// TIA Portal V20 export
FUNCTION_BLOCK "AirConditioner"   // FB349, FBD
{ S7_Optimized_Access := 'TRUE' }
// stored: AutoNumber false, MemoryReserve 100, SetENOAutomatically false
   VAR
      Var : "TypeVar";
      T : Array[1..4] of IEC_TIMER;
   END_VAR
   VAR DB_SPECIFIC
      air1Active : Bool := 1;   // air conditioner 1 scannerhousing visual measurement active
      air1InputNo : Bool := 0;   // air conditioner 1 scannerhousing visual measurement input normal
      air2Active : Bool := 1;   // air conditioner 2 scannerhousing visual measurement active
      air2InputNo : Bool := 0;   // air conditioner 2 scannerhousing visual measurement input normal
      airXrayActive : Bool := 1;   // air conditioner scannerhousing x-ray measurement active
      airXrayInputNo : Bool := 0;   // air conditioner scannerhousing x-ray measurement input normal
      airDehActive : Bool := 0;   // air dehumidifier active
      airDehInputNo : Bool := 0;   // air dehumidifier input normal open
   END_VAR
BEGIN

REGION Network 1 (SCL): air conditioner 1&2 visual measurement - config from Pc
   "G".air1Off := INT_TO_BOOL( "Param".Rd.air1Off);
   "G".air2Off := INT_TO_BOOL("Param".Rd.air2Off);
   #air1Active := INT_TO_BOOL("Param".Rd.air1Active);
   #air2Active := INT_TO_BOOL("Param".Rd.air2Active);
   #air1InputNo := INT_TO_BOOL("Param".Rd.air1InputNo);
   #air2InputNo := INT_TO_BOOL("Param".Rd.air2InputNo);
END_REGION

REGION Network 2: air conditioner 1&2 visual measurement - fault
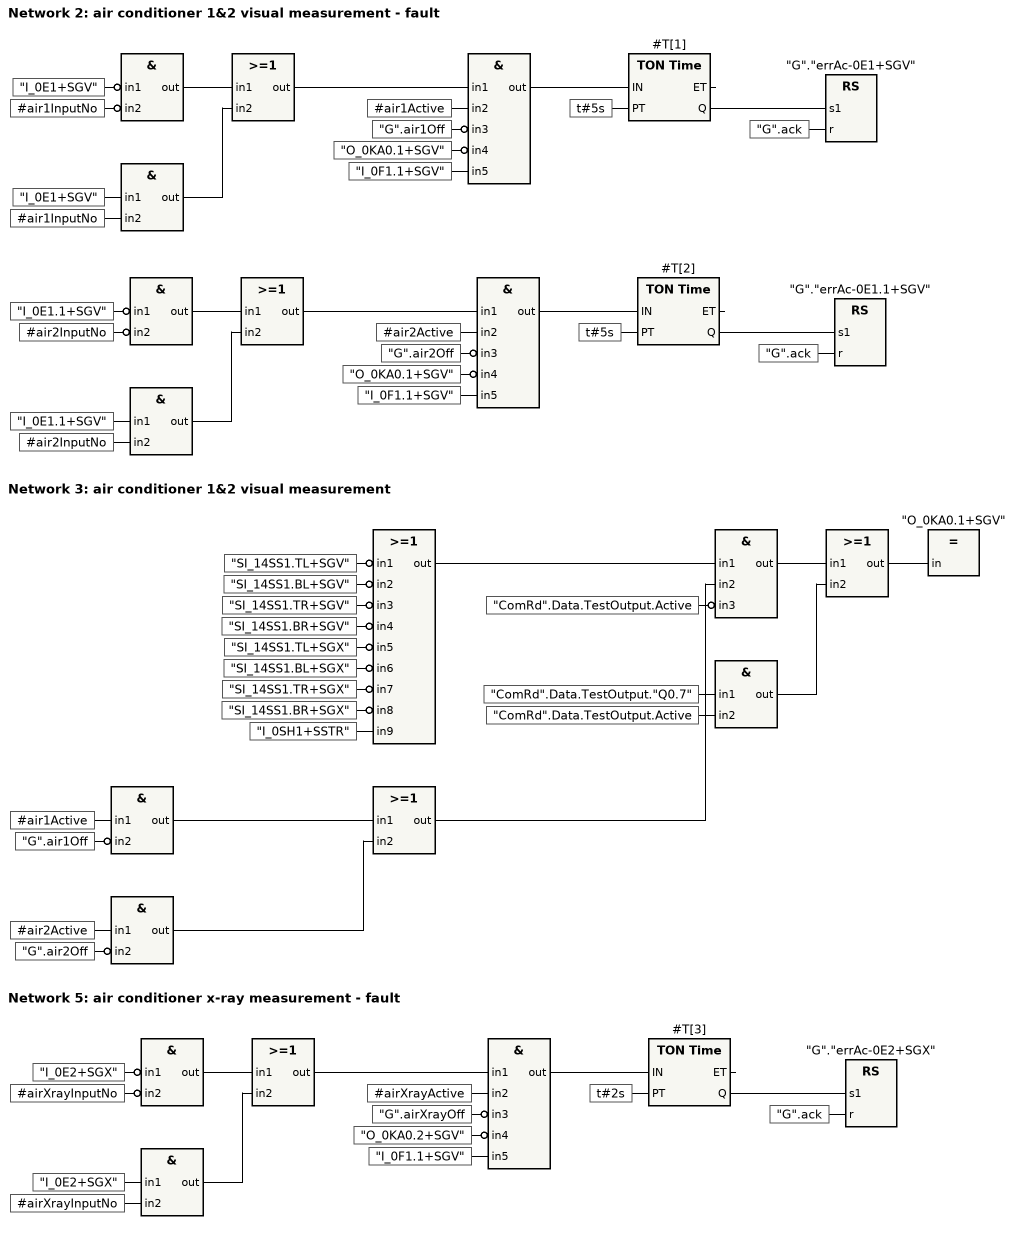
   #T[1].TON(IN := ((NOT "I_0E1+SGV" AND NOT #air1InputNo) OR ("I_0E1+SGV" AND #air1InputNo)) AND #air1Active AND NOT "G".air1Off AND NOT "O_0KA0.1+SGV" AND "I_0F1.1+SGV",
             PT := t#5s);
   IF "G".ack THEN
       "G"."errAc-0E1+SGV" := FALSE;   // RS flip-flop
   END_IF;
   IF #T[1].Q THEN "G"."errAc-0E1+SGV" := TRUE; END_IF;
   #T[2].TON(IN := ((NOT "I_0E1.1+SGV" AND NOT #air2InputNo) OR ("I_0E1.1+SGV" AND #air2InputNo)) AND #air2Active AND NOT "G".air2Off AND NOT "O_0KA0.1+SGV" AND "I_0F1.1+SGV",
             PT := t#5s);
   IF "G".ack THEN
       "G"."errAc-0E1.1+SGV" := FALSE;   // RS flip-flop
   END_IF;
   IF #T[2].Q THEN "G"."errAc-0E1.1+SGV" := TRUE; END_IF;
END_REGION

REGION Network 3: air conditioner 1&2 visual measurement
   "O_0KA0.1+SGV" := ((NOT "SI_14SS1.TL+SGV" OR NOT "SI_14SS1.BL+SGV" OR NOT "SI_14SS1.TR+SGV" OR NOT "SI_14SS1.BR+SGV" OR NOT "SI_14SS1.TL+SGX" OR NOT "SI_14SS1.BL+SGX" OR NOT "SI_14SS1.TR+SGX" OR NOT "SI_14SS1.BR+SGX" OR "I_0SH1+SSTR") AND ((#air1Active AND NOT "G".air1Off) OR (#air2Active AND NOT "G".air2Off)) AND NOT "ComRd".Data.TestOutput.Active) OR ("ComRd".Data.TestOutput."Q0.7" AND "ComRd".Data.TestOutput.Active);
END_REGION

REGION Network 4 (SCL): air conditioner x-ray measurement - config from Pc
   "G".airXrayOff := INT_TO_BOOL( "Param".Rd.airXrayOff);
   #airXrayActive := INT_TO_BOOL("Param".Rd.airXrayActive);
   #airXrayInputNo := INT_TO_BOOL("Param".Rd.airXrayInputNo);
END_REGION

REGION Network 5: air conditioner x-ray measurement - fault
   #T[3].TON(IN := ((NOT "I_0E2+SGX" AND NOT #airXrayInputNo) OR ("I_0E2+SGX" AND #airXrayInputNo)) AND #airXrayActive AND NOT "G".airXrayOff AND NOT "O_0KA0.2+SGV" AND "I_0F1.1+SGV",
             PT := t#2s);
   IF "G".ack THEN
       "G"."errAc-0E2+SGX" := FALSE;   // RS flip-flop
   END_IF;
   IF #T[3].Q THEN "G"."errAc-0E2+SGX" := TRUE; END_IF;
END_REGION

REGION Network 6: air conditioner x-ray measurement - fault
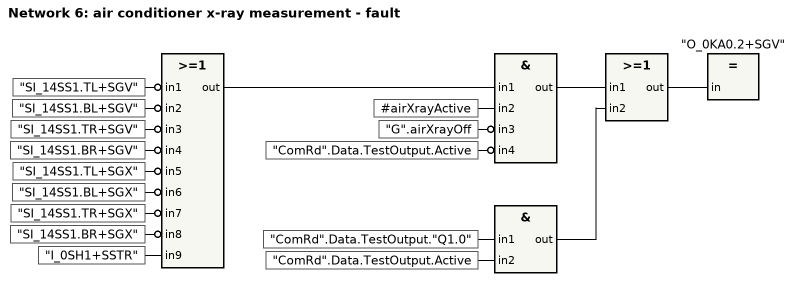
   "O_0KA0.2+SGV" := ((NOT "SI_14SS1.TL+SGV" OR NOT "SI_14SS1.BL+SGV" OR NOT "SI_14SS1.TR+SGV" OR NOT "SI_14SS1.BR+SGV" OR NOT "SI_14SS1.TL+SGX" OR NOT "SI_14SS1.BL+SGX" OR NOT "SI_14SS1.TR+SGX" OR NOT "SI_14SS1.BR+SGX" OR "I_0SH1+SSTR") AND #airXrayActive AND NOT "G".airXrayOff AND NOT "ComRd".Data.TestOutput.Active) OR ("ComRd".Data.TestOutput."Q1.0" AND "ComRd".Data.TestOutput.Active);
END_REGION
END_FUNCTION_BLOCK
